TYPE ST_ClockDefaultParameters :
STRUCT
	tTaskCycleTime	: TIME;
	tCtrlCycleTime	: TIME;
END_STRUCT
END_TYPE

(* stored: Version 1.1.0.1, ProductVersion 3.1.4024.10
   DUT ST_ClockDefaultParameters: Id {6c619834-4b10-40ab-8b26-1efe47b5b847} *)
